{attribute 'qualified_only'}
VAR_GLOBAL
	QTY: DINT;
	T1_PT: TIME := T#1S;
	Word1: WORD;
	Word3: WORD;
	CSVWORD: ARRAY[0..1] OF WORD;
	Word2: WORD;
END_VAR

(* stored: Version 1.1.0.1, ProductVersion 3.1.4024.10
   GVL GVL: Id {ac90555c-803e-4d94-8de3-f90b4c88d8f8} *)
